FUNCTION_BLOCK FILTER_MAV_DW_Test EXTENDS FB_TestSuite
VAR_INPUT
END_VAR
VAR_OUTPUT
END_VAR
VAR
END_VAR

AverageEightThenTenEqualsNine();
AverageTenThenEightEqualsNine();

METHOD AverageEightThenTenEqualsNine
VAR
	MAV : FILTER_MAV_DW;
	Result : DWORD;
	ExpectedAverage : DWORD := 9;
END_VAR
TEST('AverageEightThenTenEqualsNine');
 
MAV(X := 8, N := 2);
MAV(X := 10, Y => Result);
 
AssertEquals(Expected := ExpectedAverage,
             Actual := Result,
             Message := 'The calculation is not correct');
 
TEST_FINISHED();
END_METHOD

METHOD AverageTenThenEightEqualsNine
VAR
	MAV : FILTER_MAV_DW;
	Result : DWORD;
	ExpectedAverage : DWORD := 9;
END_VAR
TEST('AverageTenThenEightEqualsNine');
 
MAV(X := 10, N := 2);
MAV(X := 8, Y => Result);
 
AssertEquals(Expected := ExpectedAverage,
             Actual := Result,
             Message := 'The calculation is not correct');
 
TEST_FINISHED();
END_METHOD

END_FUNCTION_BLOCK

(* stored: Version 1.1.0.1, ProductVersion 3.1.4024.9
   POU FILTER_MAV_DW_Test: Id {9ae2d138-1421-4906-88bd-6a21dc08490c}, SpecialFunc None
   Method AverageEightThenTenEqualsNine: Id {ddf0513e-bd3c-42d5-b90b-a90ff4cb74a5}
   Method AverageTenThenEightEqualsNine: Id {8a8b84d5-13c5-450e-b7f8-032e2929635f} *)
